// Base interface for an operator.
INTERFACE I_Operator EXTENDS I_Object

END_INTERFACE

(* stored: Version 1.1.0.1, ProductVersion 3.1.4024.4
   Itf I_Operator: Id {ee3147cf-4b2d-48de-a79b-65b9016a509c} *)
